TYPE Room_Ctx_Io_In :
STRUCT
	rTemperature		: REAL;
END_STRUCT
END_TYPE

(* stored: Version 1.1.0.1
   DUT Room_Ctx_Io_In: Id {6a9e75f9-cfe2-41a6-a480-be45bb9be67b} *)
